{attribute addProperty BoxType "BK1120-0000-0018"}
{attribute addProperty Id "Term_378_KL1002KL1002_D229A9CA00"}
{attribute addProperty CRC "3968576433"}
{attribute addProperty SizeInBites "0"}
{attribute addProperty SizeInBytes "0"}
TYPE A_0005_BK1120_0000_0018_EC8BABB1 EXTENDS BK1120_4487A81F :
STRUCT
	{attribute addProperty Name "Term_378_KL1002"}
	Term_378_KL1002 : KL1002_D229A9CA;
END_STRUCT
END_TYPE

(* stored: Version 1.2.0.0, ProductVersion 3.1.4024.9
   DUT A_0005_BK1120_0000_0018_EC8BABB1: Id {6361de78-257b-41bd-87cc-e106ec9ce6de} *)
